FUNCTION_BLOCK ValidateFunctionsTest EXTENDS TcUnit.FB_TestSuite
VAR
END_VAR

StringBeginsWithAnyFunction();
StringEndsWithAnyFunction();

METHOD StringBeginsWithAnyFunction : BOOL
VAR
	test : T_MaxString := 'this is test string';
END_VAR
TcUnit.TEST('String begins with');

AssertEquals_BOOL(
	Expected := FALSE,
	Actual := StringBeginsWithAny(test, 'nothing'),
	Message := 'Should return FALSE because string does not begin with checked value');

AssertEquals_BOOL(
	Expected := TRUE,
	Actual := StringBeginsWithAny(test, 'this'),
	Message := 'Should return TRUE because string begins with checked value');

TEST_FINISHED();
END_METHOD

METHOD StringEndsWithAnyFunction : BOOL
VAR
	test : T_MaxString := 'this is test string';
END_VAR
TcUnit.TEST('String ends with');

AssertEquals_BOOL(
	Expected := FALSE,
	Actual := StringBeginsWithAny(test, 'nothing'),
	Message := 'Should return FALSE because string does not end with checked value');

AssertEquals_BOOL(
	Expected := TRUE,
	Actual := StringEndsWithAny(test, 'string'),
	Message := 'Should return TRUE because string ends with checked value');

TEST_FINISHED();
END_METHOD

END_FUNCTION_BLOCK

(* stored: Version 1.1.0.1, ProductVersion 3.1.4024.15
   POU ValidateFunctionsTest: Id {cb16a091-8ccb-0ed8-19c5-6ad231cd9912}, SpecialFunc None
   Method StringBeginsWithAnyFunction: Id {800b0c27-0a41-0ee5-0ced-ca7be9a08bff}
   Method StringEndsWithAnyFunction: Id {1a96034c-2cd2-0bb9-2016-37253a64c0e9} *)
